TYPE InertiaEmulation_Struct_EAP :
UNION
		Value : INT;
		Bits : Bits_InertiaEmulation_EAP;
END_UNION
END_TYPE

(* stored: Version 1.1.0.1, ProductVersion 3.1.4022.18
   DUT InertiaEmulation_Struct_EAP: Id {936504c1-b387-4f7e-8aa6-1e5295d18753} *)
